TYPE MC_ErrorID_Udint : UDINT; END_TYPE

(* stored: Version 1.1.0.1, ProductVersion 3.1.4024.12
   DUT MC_ErrorID_Udint: Id {23c9f0e6-0ae1-4520-92a7-95cbfc91b275} *)
